{attribute 'qualified_only'}
VAR_GLOBAL
END_VAR

(* stored: Version 1.1.0.1, ProductVersion 3.1.4022.18
   GVL GVL_1: Id {af1f44fe-2131-4234-9e37-3513fd886410} *)
